PROGRAM EM04_PlacingArea_3
VAR
//----Motor-----
	// Box Placing Roller Conveyor 3	
	FB_BoxPlacingRollerConv_3			: MotorManagement;
	stBoxPlacingRollerConv_3			: stMotor;
	BoxPlacingRollerConv_3_ErrorID		: UINT;
	BoxPlacingRollerConv_3_Error		: BOOL;
	bFL_BoxPlacingRollerConv_3_Forward	: BOOL;
	bFL_BoxPlacingRollerConv_3_Reverse	: BOOL;
END_VAR

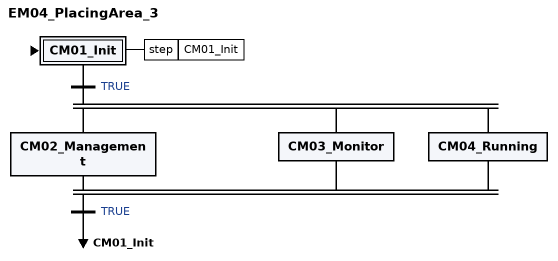
INITIAL_STEP CM01_Init:
    CM01_Init(N);  // step action
END_STEP
TRANSITION FROM CM01_Init TO (CM02_Management, CM03_Monitor, CM04_Running)
    := TRUE;
END_TRANSITION
STEP CM02_Management:
END_STEP
STEP CM03_Monitor:
END_STEP
STEP CM04_Running:
END_STEP
TRANSITION FROM (CM02_Management, CM03_Monitor, CM04_Running) TO CM01_Init
    := TRUE;
END_TRANSITION

ACTION CM01_Init:

END_ACTION

ACTION CM02_Management:
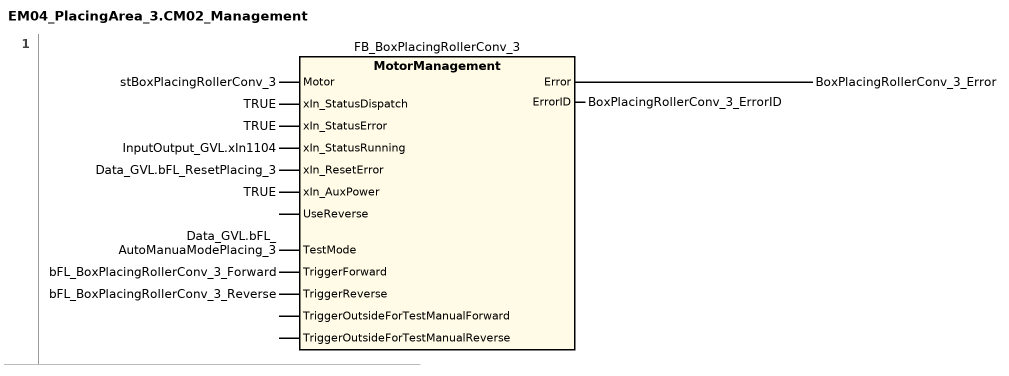
// NETWORK 1
FB_BoxPlacingRollerConv_3(
    Motor := stBoxPlacingRollerConv_3,
    xIn_StatusDispatch := TRUE,
    xIn_StatusError := TRUE,
    xIn_StatusRunning := InputOutput_GVL.xIn1104,
    xIn_ResetError := Data_GVL.bFL_ResetPlacing_3,
    xIn_AuxPower := TRUE,
    TestMode := Data_GVL.bFL_AutoManuaModePlacing_3,
    TriggerForward := bFL_BoxPlacingRollerConv_3_Forward,
    TriggerReverse := bFL_BoxPlacingRollerConv_3_Reverse,
    ErrorID => BoxPlacingRollerConv_3_ErrorID); // MotorManagement
BoxPlacingRollerConv_3_Error := FB_BoxPlacingRollerConv_3.Error;
END_ACTION

ACTION CM03_Monitor:
// NETWORK 1
END_ACTION

ACTION CM04_Running:
// NETWORK 1
END_ACTION

END_PROGRAM

(* stored: Version 1.1.0.1, ProductVersion 3.1.4024.9
   POU EM04_PlacingArea_3: Id {59d8dee2-b50a-4354-8ed8-a4469c44a0eb}, SpecialFunc None
   Action CM01_Init: Id {ac53e07a-d766-4c91-a110-4a97d5863136}
   Action CM02_Management: Id {fce01ecb-1dce-40b4-a923-f0ec23d35ea2}
   Action CM03_Monitor: Id {5537a70e-6ce0-4d03-8528-22743b9fba23}
   Action CM04_Running: Id {f74debe0-1e5d-4416-bc8d-9870e6097fad} *)
